// TIA Portal project "TCP IP_V13_SP1" (V13)

(* hardware
DEVICE "S7-1200 station_1"  S7-1200 Station
   slot 0: "Rack_0"  Rack  V1.0
   slot 1: "PLC_1"  CPU 1214C DC/DC/DC  6ES7 214-1AG40-0XB0  V4.1
   slot 3: "AQ 1x12BIT_1"  6ES7 232-4HA30-0XB0  V1.0
DEVICE "S7-1200 station_2"  S7-1200 Station
   slot 0: "Rack_0"  Rack  V1.0
   slot 1: "PLC_2"  CPU 1214C DC/DC/DC  6ES7 214-1AG40-0XB0  V4.1
   slot 3: "AQ 1x12BIT_1"  6ES7 232-4HA30-0XB0  V1.0
*)

// ===== PLC "PLC_1"  CPU 1214C DC/DC/DC =====

VAR_GLOBAL   // PLC tag table "Default tag table"
   "Tag_1" AT %I0.0 : Bool;
END_VAR

DATA_BLOCK "MyDataToSend"   // DB1
{ S7_Optimized_Access := 'FALSE' }
VERSION : 0.1
   VAR
      Data : Struct
      END_STRUCT;
      Done : Bool;
      Busy : Bool;
      Data1 : UInt;
   END_VAR
BEGIN
END_DATA_BLOCK

DATA_BLOCK "MyDataToReceive"   // DB6
{ S7_Optimized_Access := 'FALSE' }
VERSION : 0.1
   VAR
      Data : Struct
      END_STRUCT;
      Done : Bool;
      Busy : Bool;
      Data1 : UInt;
   END_VAR
BEGIN
END_DATA_BLOCK

// folder: System blocks/Program resources

DATA_BLOCK "PLC_1_Send_DB"   // DB3
{ S7_Optimized_Access := 'FALSE' }
AUTHOR : SIMATIC
FAMILY : MC7Plus
NAME : TC_IP_v4
VERSION : 1.0
// stored: InstanceOfName ?
"?"
BEGIN
END_DATA_BLOCK

DATA_BLOCK "CPU SEND_Connection_DB"   // DB4
{ S7_Optimized_Access := 'FALSE' }
AUTHOR : SIMATIC
FAMILY : MC7Plus
NAME : TCON_Prm
VERSION : 1.0
// stored: InstanceOfName ?
"?"
BEGIN
   LOCAL_TSAP_ID[1] := B#16#00;
   LOCAL_TSAP_ID[2] := B#16#00;
   LOCAL_TSAP_ID[3] := B#16#00;
   LOCAL_TSAP_ID[4] := B#16#00;
   LOCAL_TSAP_ID[5] := B#16#00;
   LOCAL_TSAP_ID[6] := B#16#00;
   LOCAL_TSAP_ID[7] := B#16#00;
   LOCAL_TSAP_ID[8] := B#16#00;
   LOCAL_TSAP_ID[9] := B#16#00;
   LOCAL_TSAP_ID[10] := B#16#00;
   LOCAL_TSAP_ID[11] := B#16#00;
   LOCAL_TSAP_ID[12] := B#16#00;
   LOCAL_TSAP_ID[13] := B#16#00;
   LOCAL_TSAP_ID[14] := B#16#00;
   LOCAL_TSAP_ID[15] := B#16#00;
   LOCAL_TSAP_ID[16] := B#16#00;
   REM_TSAP_ID[1] := B#16#07;
   REM_TSAP_ID[2] := B#16#D0;
   REM_TSAP_ID[3] := B#16#00;
   REM_TSAP_ID[4] := B#16#00;
   REM_TSAP_ID[5] := B#16#00;
   REM_TSAP_ID[6] := B#16#00;
   REM_TSAP_ID[7] := B#16#00;
   REM_TSAP_ID[8] := B#16#00;
   REM_TSAP_ID[9] := B#16#00;
   REM_TSAP_ID[10] := B#16#00;
   REM_TSAP_ID[11] := B#16#00;
   REM_TSAP_ID[12] := B#16#00;
   REM_TSAP_ID[13] := B#16#00;
   REM_TSAP_ID[14] := B#16#00;
   REM_TSAP_ID[15] := B#16#00;
   REM_TSAP_ID[16] := B#16#00;
   REM_SUBNET_ID[1] := 0;
   REM_SUBNET_ID[2] := 0;
   REM_SUBNET_ID[3] := 0;
   REM_SUBNET_ID[4] := 0;
   REM_SUBNET_ID[5] := 0;
   REM_SUBNET_ID[6] := 0;
   REM_STADDR[1] := 140;
   REM_STADDR[2] := 80;
   REM_STADDR[3] := 0;
   REM_STADDR[4] := 1;
   REM_STADDR[5] := 0;
   REM_STADDR[6] := 0;
   NEXT_STADDR[1] := B#16#0;
   NEXT_STADDR[2] := B#16#0;
   NEXT_STADDR[3] := B#16#0;
   NEXT_STADDR[4] := B#16#0;
   NEXT_STADDR[5] := B#16#0;
   NEXT_STADDR[6] := B#16#0;
END_DATA_BLOCK

// folder: (top level)

FUNCTION "SendEthernet" : Void   // FC1, LAD
{ S7_Optimized_Access := 'FALSE' }
VERSION : 0.1
BEGIN

REGION Network 1
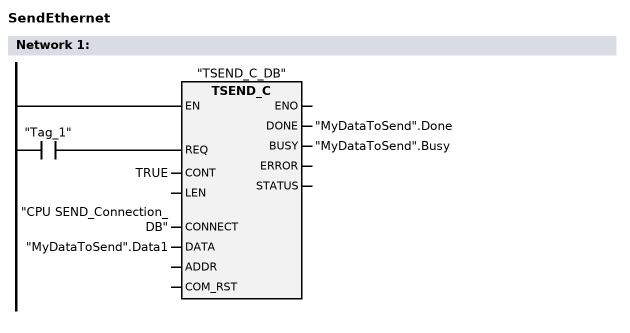
   "TSEND_C_DB"(REQ := "Tag_1",   // TSEND_C
                CONT := TRUE,
                CONNECT := "CPU SEND_Connection_DB",
                DATA := "MyDataToSend".Data1,
                DONE => "MyDataToSend".Done,
                BUSY => "MyDataToSend".Busy);
END_REGION
END_FUNCTION

FUNCTION "ReceiveEthernet" : Void   // FC2, LAD
{ S7_Optimized_Access := 'FALSE' }
VERSION : 0.1
BEGIN

REGION Network 1
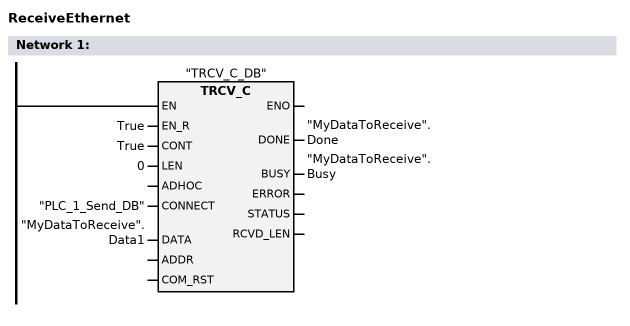
   "TRCV_C_DB"(EN_R := True,   // TRCV_C
               CONT := True,
               LEN := 0,
               CONNECT := "PLC_1_Send_DB",
               DATA := "MyDataToReceive".Data1,
               DONE => "MyDataToReceive".Done,
               BUSY => "MyDataToReceive".Busy);
END_REGION
END_FUNCTION

ORGANIZATION_BLOCK "Main"   // OB1, LAD, ProgramCycle
TITLE = "Main Program Sweep (Cycle)"
{ S7_Optimized_Access := 'FALSE' }
VERSION : 0.1
BEGIN

REGION Network 1: Send
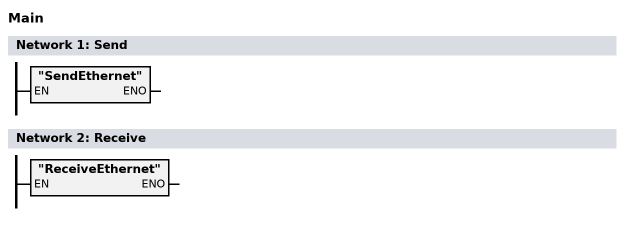
   RUNG wire#powerrail
      "SendEthernet"()
   END_RUNG
   // the same network as SCL:
   "SendEthernet"();
END_REGION

REGION Network 2: Receive
   RUNG wire#powerrail
      "ReceiveEthernet"()
   END_RUNG
   // the same network as SCL:
   "ReceiveEthernet"();
END_REGION
END_ORGANIZATION_BLOCK

// ===== PLC "PLC_2"  CPU 1214C DC/DC/DC =====

VAR_GLOBAL   // PLC tag table "Default tag table"
   "Tag_1" AT %I0.0 : Bool;
END_VAR

DATA_BLOCK "MyDataToReceive"   // DB1
{ S7_Optimized_Access := 'FALSE' }
VERSION : 0.1
   VAR
      DATA : Struct
      END_STRUCT;
      Done : Bool;
      Busy : Bool;
      Data1 : UInt;
   END_VAR
BEGIN
END_DATA_BLOCK

DATA_BLOCK "MyDataToSend"   // DB4
{ S7_Optimized_Access := 'FALSE' }
VERSION : 0.1
   VAR
      Data : Struct
      END_STRUCT;
      Done : Bool;
      Busy : Bool;
      Data1 : UInt;
   END_VAR
BEGIN
END_DATA_BLOCK

// folder: System blocks/Program resources

DATA_BLOCK "PLC_2_Receive_DB"   // DB2
{ S7_Optimized_Access := 'FALSE' }
AUTHOR : SIMATIC
FAMILY : MC7Plus
NAME : TC_IP_v4
VERSION : 1.0
// stored: InstanceOfName ?
"?"
BEGIN
END_DATA_BLOCK

DATA_BLOCK "PLC_2_Send_DB"   // DB6
{ S7_Optimized_Access := 'FALSE' }
AUTHOR : SIMATIC
FAMILY : MC7Plus
NAME : TC_IP_v4
VERSION : 1.0
// stored: InstanceOfName ?
"?"
BEGIN
END_DATA_BLOCK

// folder: (top level)

FUNCTION "SendEthernet" : Void   // FC1, LAD
{ S7_Optimized_Access := 'FALSE' }
VERSION : 0.1
BEGIN

REGION Network 1
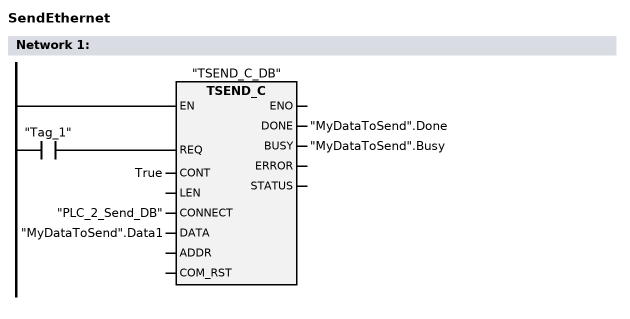
   "TSEND_C_DB"(REQ := "Tag_1",   // TSEND_C
                CONT := True,
                CONNECT := "PLC_2_Send_DB",
                DATA := "MyDataToSend".Data1,
                DONE => "MyDataToSend".Done,
                BUSY => "MyDataToSend".Busy);
END_REGION
END_FUNCTION

FUNCTION "ReceiveEthernet" : Void   // FC2, LAD
{ S7_Optimized_Access := 'FALSE' }
VERSION : 0.1
BEGIN

REGION Network 1
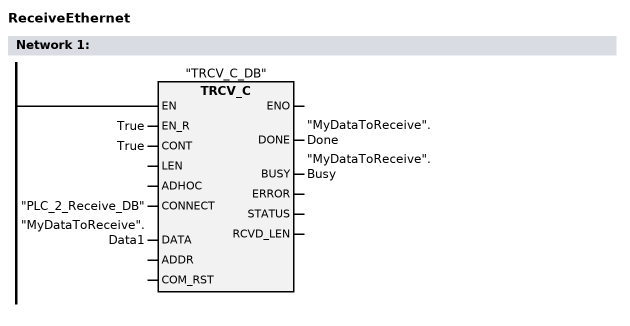
   "TRCV_C_DB"(EN_R := True,   // TRCV_C
               CONT := True,
               CONNECT := "PLC_2_Receive_DB",
               DATA := "MyDataToReceive".Data1,
               DONE => "MyDataToReceive".Done,
               BUSY => "MyDataToReceive".Busy);
END_REGION
END_FUNCTION

ORGANIZATION_BLOCK "Main"   // OB1, LAD, ProgramCycle
TITLE = "Main Program Sweep (Cycle)"
{ S7_Optimized_Access := 'FALSE' }
VERSION : 0.1
BEGIN

REGION Network 1: Receive
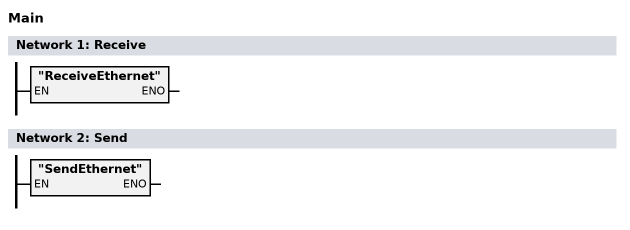
   RUNG wire#powerrail
      "ReceiveEthernet"()
   END_RUNG
   // the same network as SCL:
   "ReceiveEthernet"();
END_REGION

REGION Network 2: Send
   RUNG wire#powerrail
      "SendEthernet"()
   END_RUNG
   // the same network as SCL:
   "SendEthernet"();
END_REGION
END_ORGANIZATION_BLOCK